PROGRAM FC3
VAR
END_VAR

END_PROGRAM

(* stored: Version 1.1.0.1, ProductVersion 3.1.4022.12
   POU FC3: Id {0e42956f-4f7f-45d6-9596-8a90c0d9b087}, SpecialFunc None *)
